// TIA Portal V17 export
// export: Created 2025-03-07T09:19:05.7984013Z, ExportSetting WithDefaults, DisplayName Totally Integrated Automation Portal, DisplayVersion V17 Update 8, DisplayName TIA Portal Openness, DisplayVersion V17 Update 8, DisplayName TIA Portal Version Control Interface, DisplayVersion V17, DisplayName SINAMICS Startdrive Advanced, DisplayVersion V17 SP2, DisplayName SINAMICS Startdrive G110M, G120, G120C, G120D, G120P, G115D, DisplayVersion V17 SP2, DisplayName SINAMICS Startdrive G130, G150, S120, S150, SINAMICS MV, S210, DisplayVersion V17 SP2, DisplayName STEP 7 Professional, DisplayVersion V17 Update 8, DisplayName SINUMERIK ONE STEP 7 Toolbox, DisplayVersion V17 Update 12, DisplayName SINUMERIK 840D sl STEP 7 Toolbox, DisplayVersion V17 Update 12, DisplayName STEP 7 Safety, DisplayVersion V17 Update 6, DisplayName WinCC Advanced, DisplayVersion V17 Update 8
DATA_BLOCK "DB16701_OPC_UA_MASTER_MACHINE"   // DB16701
{ S7_Optimized_Access := 'FALSE' }
VERSION : 0.1
// stored: AutoNumber false, DBAccessibleFromOPCUA true, DBAccessibleFromWebserver true, IsOnlyStoredInLoadMemory false, IsWriteProtectedInAS false
   VAR
      GENERAL { ExternalWritable := 'False'} : Struct
         ID { ExternalWritable := 'False'} : Struct
            LINE { ExternalWritable := 'False'} : Int;   // GENERAL INFORMATION: PRODUCTION LINE IDENTIFICATION
            MACHINE { ExternalWritable := 'False'} : Int;   // GENERAL INFORMATION: PRODUCTION MACHINE IDENTIFICATION
            PLC { ExternalWritable := 'False'} : Int;   // GENERAL INFORMATION: PRODUCTION PLC IDENTIFICATION (POWDER PLC = 1 / MACHINE PLC = 2 / CELL PLC = 3)
         END_STRUCT;
         WORKER { ExternalWritable := 'False'} : Struct
            ID { ExternalWritable := 'False'} : Int;
         END_STRUCT;
         PART_TRACKING { ExternalWritable := 'False'} : Struct
            UNIT_01 { ExternalWritable := 'False'} : Struct
               STA1 { ExternalWritable := 'False'} : Struct
                  DMC { ExternalWritable := 'False'} : Array[0..63] of Char;   // DMC PART NUMBER IN UNIT 01 STATION 1
                  FIXTURE_NUMBER { ExternalWritable := 'False'} : Int;   // FIXTURE NUMBER IN UNIT 01 STATION 1
               END_STRUCT;
               STA2 { ExternalWritable := 'False'} : Struct
                  DMC { ExternalWritable := 'False'} : Array[0..63] of Char;   // DMC PART NUMBER IN UNIT 01 STATION 2
                  FIXTURE_NUMBER { ExternalWritable := 'False'} : Int;   // FIXTURE NUMBER IN UNIT 01 STATION 2
               END_STRUCT;
               STA3 { ExternalWritable := 'False'} : Struct
                  DMC { ExternalWritable := 'False'} : Array[0..63] of Char;   // DMC PART NUMBER IN UNIT 01 STATION 3
                  FIXTURE_NUMBER { ExternalWritable := 'False'} : Int;   // FIXTURE NUMBER IN UNIT 01 STATION 3
               END_STRUCT;
               STA4 { ExternalWritable := 'False'} : Struct
                  DMC { ExternalWritable := 'False'} : Array[0..63] of Char;   // DMC PART NUMBER IN UNIT 01 STATION 4
                  FIXTURE_NUMBER { ExternalWritable := 'False'} : Int;   // FIXTURE NUMBER IN UNIT 01 STATION 4
               END_STRUCT;
            END_STRUCT;
            UNIT_02 { ExternalWritable := 'False'} : Struct
               STA1 { ExternalWritable := 'False'} : Struct
                  DMC { ExternalWritable := 'False'} : Array[0..63] of Char;   // DMC PART NUMBER IN UNIT 02 STATION 1
                  FIXTURE_NUMBER { ExternalWritable := 'False'} : Int;   // FIXTURE NUMBER IN UNIT 02 STATION 1
               END_STRUCT;
               STA2 { ExternalWritable := 'False'} : Struct
                  DMC { ExternalWritable := 'False'} : Array[0..63] of Char;   // DMC PART NUMBER IN UNIT 02 STATION 2
                  FIXTURE_NUMBER { ExternalWritable := 'False'} : Int;   // FIXTURE NUMBER IN UNIT 02 STATION 2
               END_STRUCT;
               STA3 { ExternalWritable := 'False'} : Struct
                  DMC { ExternalWritable := 'False'} : Array[0..63] of Char;   // DMC PART NUMBER IN UNIT 02 STATION 3
                  FIXTURE_NUMBER { ExternalWritable := 'False'} : Int;   // FIXTURE NUMBER IN UNIT 02 STATION 3
               END_STRUCT;
               STA4 { ExternalWritable := 'False'} : Struct
                  DMC { ExternalWritable := 'False'} : Array[0..63] of Char;   // DMC PART NUMBER IN UNIT 02 STATION 4
                  FIXTURE_NUMBER { ExternalWritable := 'False'} : Int;   // FIXTURE NUMBER IN UNIT 02 STATION 4
               END_STRUCT;
            END_STRUCT;
         END_STRUCT;
         SHARED_AIR_EXTRACTION { ExternalWritable := 'False'} : Struct
            INPUT_KELLER_PRESSURE { ExternalWritable := 'False'} : Real;   // MACHINE AIR EXTRACTION INPUT KELLER PRESSURE VALUE (Bar)
            PRESSURE_DIFFERENCE_FILTER { ExternalWritable := 'False'} : Real;   // MACHINE AIR EXTRACTION PRESSURE DIFFERENCE IN FILTER VALUE (Bar)
         END_STRUCT;
      END_STRUCT;
      UNIT_01 { ExternalWritable := 'False'} : Struct
         MACHINE { ExternalWritable := 'False'} : Struct
            PNEUMATIC_STATE { ExternalWritable := 'False'} : Bool;   // UNIT 01 PNEUMATIC STATE: CORRECT WORKING (NO FAULTS)
            TEMPERATURE { ExternalWritable := 'False'} : Struct
               DISC_SURFACE { ExternalWritable := 'False'} : Real;   // UNIT 01 MACHINE TEMPERATURE: DISC SURFACE (ºC)
               AMBIENT_PYROMETER { ExternalWritable := 'False'} : Real;   // UNIT 01 MACHINE TEMPERATURE: AMBIENT PYROMETER (ºC)
               EMISIVITY_CURVE { ExternalWritable := 'False'} : Real;   // UNIT 01 MACHINE TEMPERATURE: EMISIVITY CURVE (¿?¿?¿?¿?¿?)
            END_STRUCT;
            COOLING_SYSTEM { ExternalWritable := 'False'} : Struct
               INPUT_FLOW { ExternalWritable := 'False'} : Real;   // UNIT 01 COOLING SYSTEM INPUT FLOW VALUE (l/min)
               INPUT_TEMPERATURE { ExternalWritable := 'False'} : Real;   // UNIT 01 COOLING SYSTEM INPUT TEMPERATURE VALUE (ºC)
               OUTPUT_FLOW { ExternalWritable := 'False'} : Real;   // UNIT 01 COOLING SYSTEM OUTPUT FLOW VALUE (l/min)
               OUTPUT_TEMPERATURE { ExternalWritable := 'False'} : Real;   // UNIT 01 COOLING SYSTEM OUTPUT TEMPERATURE VALUE (ºC)
               LASER_HEAD_FLOW { ExternalWritable := 'False'} : Real;   // UNIT 01 COOLING SYSTEM LASER HEAD FLOW VALUE (l/min)
               LASER_HEAD_TEMPERATURE { ExternalWritable := 'False'} : Real;   // UNIT 01 COOLING SYSTEM LASER HEAD TEMPERATURE VALUE (ºC)
               LASER_FLOW { ExternalWritable := 'False'} : Real;   // UNIT 01 COOLING SYSTEM LASER FLOW VALUE (l/min)
               LASER_TEMPERATURE { ExternalWritable := 'False'} : Real;   // UNIT 01 COOLING SYSTEM LASER TEMPERATURE VALUE (ºC)
               NOZZLE_FLOW { ExternalWritable := 'False'} : Real;   // UNIT 01 COOLING SYSTEM LASER NOZZLE FLOW VALUE (l/min)
               NOZZLE_TEMPERATURE { ExternalWritable := 'False'} : Real;   // UNIT 01 COOLING SYSTEM LASER NOZZLE TEMPERATURE VALUE (ºC)
               SHIELD_FLOW { ExternalWritable := 'False'} : Real;   // UNIT 01 COOLING SYSTEM SHIELD FLOW VALUE (l/min)
               SHIELD_TEMPERATURE { ExternalWritable := 'False'} : Real;   // UNIT 01 COOLING SYSTEM SHIELD TEMPERATURE VALUE (ºC)
            END_STRUCT;
            AIR_EXTRACTION { ExternalWritable := 'False'} : Struct
               OUTPUT_PRESSURE { ExternalWritable := 'False'} : Real;   // UNIT 01 AIR EXTRACTION OUTPUT PRESSURE VALUE (Bar)
               ST3_PRESSURE { ExternalWritable := 'False'} : Real;   // UNIT 01 STA 3 PRESSURE CONTROL
            END_STRUCT;
            POSITIONS { ExternalWritable := 'False'} : Struct
               CN { ExternalWritable := 'False'} : Struct
                  X13 { ExternalWritable := 'False'} : Real;   // UNIT 01 AXIS X13 POSITION VALUE
                  Z13 { ExternalWritable := 'False'} : Real;   // UNIT 01 AXIS Z13 POSITION VALUE
               END_STRUCT;
               LASER_HEAD { ExternalWritable := 'False'} : Struct
                  RADIAL_ANGLE { ExternalWritable := 'False'} : Bool;   // UNIT 01 LASER HEAD RADIAL ANGLE ADVANCED
                  TANGENTIAL_ANGLE { ExternalWritable := 'False'} : Bool;   // UNIT 01 LASER HEAD TANGENTIAL ANGLE ADVANCED
               END_STRUCT;
            END_STRUCT;
            SPEED { ExternalWritable := 'False'} : Struct
               X13 { ExternalWritable := 'False'} : Real;   // UNIT 01 AXIS X13 SPEED VALUE (mm/min)
               C13 { ExternalWritable := 'False'} : Real;   // UNIT 01 AXIS C13 SPEED VALUE (º/min)
               PROCESS_SETPOINT { ExternalWritable := 'False'} : Real;   // UNIT 01 SPEED PROCESS SETPOINT (mm/min)
            END_STRUCT;
            NOZZLE { ExternalWritable := 'False'} : Struct
               SHIELD_GAS_FLOW { ExternalWritable := 'False'} : Real;   // UNIT 01 SHIELD GAS FLOW VALUE (nl/min)
            END_STRUCT;
         END_STRUCT;
         PROCESS { ExternalWritable := 'False'} : Struct
            STATION_1_RUNNING { ExternalWritable := 'False'} : Bool;   // UNIT 01 CLADDING STATION 1 RUNNING
            STATION_2_RUNNING { ExternalWritable := 'False'} : Bool;   // UNIT 01 CLADDING STATION 2 RUNNING
            STATION_3_RUNNING { ExternalWritable := 'False'} : Bool;   // UNIT 01 CLADDING STATION 3 RUNNING
            STATION_4_RUNNING { ExternalWritable := 'False'} : Bool;   // UNIT 01 CLADDING STATION 4 RUNNING
            LASER_ON { ExternalWritable := 'False'} : Bool;   // UNIT 01 LASER ON
            FIXTURE_SEALING { ExternalWritable := 'False'} : Bool;   // UNIT 01 FIXTURE SEALING CLOSED
         END_STRUCT;
      END_STRUCT;
      UNIT_02 { ExternalWritable := 'False'} : Struct
         MACHINE { ExternalWritable := 'False'} : Struct
            PNEUMATIC_STATE { ExternalWritable := 'False'} : Bool;   // UNIT 02 PNEUMATIC STATE: CORRECT WORKING (NO FAULTS)
            TEMPERATURE { ExternalWritable := 'False'} : Struct
               DISC_SURFACE { ExternalWritable := 'False'} : Real;   // UNIT 02 MACHINE TEMPERATURE: DISC SURFACE (ºC)
               AMBIENT_PYROMETER { ExternalWritable := 'False'} : Real;   // UNIT 02 MACHINE TEMPERATURE: AMBIENT PYROMETER (ºC)
               EMISIVITY_CURVE { ExternalWritable := 'False'} : Real;   // UNIT 02 MACHINE TEMPERATURE: EMISIVITY CURVE (¿?¿?¿?¿?¿?)
            END_STRUCT;
            COOLING_SYSTEM { ExternalWritable := 'False'} : Struct
               INPUT_FLOW { ExternalWritable := 'False'} : Real;   // UNIT 02 COOLING SYSTEM INPUT FLOW VALUE (l/min)
               INPUT_TEMPERATURE { ExternalWritable := 'False'} : Real;   // UNIT 02 COOLING SYSTEM INPUT TEMPERATURE VALUE (ºC)
               OUTPUT_FLOW { ExternalWritable := 'False'} : Real;   // UNIT 02 COOLING SYSTEM OUTPUT FLOW VALUE (l/min)
               OUTPUT_TEMPERATURE { ExternalWritable := 'False'} : Real;   // UNIT 02 COOLING SYSTEM OUTPUT TEMPERATURE VALUE (ºC)
               LASER_HEAD_FLOW { ExternalWritable := 'False'} : Real;   // UNIT 02 COOLING SYSTEM LASER HEAD FLOW VALUE (l/min)
               LASER_HEAD_TEMPERATURE { ExternalWritable := 'False'} : Real;   // UNIT 02 COOLING SYSTEM LASER HEAD TEMPERATURE VALUE (ºC)
               LASER_FLOW { ExternalWritable := 'False'} : Real;   // UNIT 02 COOLING SYSTEM LASER FLOW VALUE (l/min)
               LASER_TEMPERATURE { ExternalWritable := 'False'} : Real;   // UNIT 02 COOLING SYSTEM LASER TEMPERATURE VALUE (ºC)
               NOZZLE_FLOW { ExternalWritable := 'False'} : Real;   // UNIT 02 COOLING SYSTEM LASER NOZZLE FLOW VALUE (l/min)
               NOZZLE_TEMPERATURE { ExternalWritable := 'False'} : Real;   // UNIT 02 COOLING SYSTEM LASER NOZZLE TEMPERATURE VALUE (ºC)
               SHIELD_FLOW { ExternalWritable := 'False'} : Real;   // UNIT 02 COOLING SYSTEM SHIELD FLOW VALUE (l/min)
               SHIELD_TEMPERATURE { ExternalWritable := 'False'} : Real;   // UNIT 02 COOLING SYSTEM SHIELD TEMPERATURE VALUE (ºC)
            END_STRUCT;
            AIR_EXTRACTION { ExternalWritable := 'False'} : Struct
               OUTPUT_PRESSURE { ExternalWritable := 'False'} : Real;   // UNIT 02 AIR EXTRACTION OUTPUT PRESSURE VALUE (Bar)
               ST3_PRESSURE { ExternalWritable := 'False'} : Real;   // UNIT 02 STA 3 PRESSURE CONTROL
            END_STRUCT;
            POSITIONS { ExternalWritable := 'False'} : Struct
               CN { ExternalWritable := 'False'} : Struct
                  X23 { ExternalWritable := 'False'} : Real;   // UNIT 02 AXIS X23 POSITION VALUE
                  Z23 { ExternalWritable := 'False'} : Real;   // UNIT 02 AXIS Z23 POSITION VALUE
               END_STRUCT;
               LASER_HEAD { ExternalWritable := 'False'} : Struct
                  RADIAL_ANGLE { ExternalWritable := 'False'} : Bool;   // UNIT 02 LASER HEAD RADIAL ANGLE ADVANCED
                  TANGENTIAL_ANGLE { ExternalWritable := 'False'} : Bool;   // UNIT 02 LASER HEAD TANGENTIAL ANGLE ADVANCED
               END_STRUCT;
            END_STRUCT;
            SPEED { ExternalWritable := 'False'} : Struct
               X23 { ExternalWritable := 'False'} : Real;   // UNIT 02 AXIS X23 SPEED VALUE (mm/min)
               C23 { ExternalWritable := 'False'} : Real;   // UNIT 02 AXIS C23 SPEED VALUE (º/min)
               PROCESS_SETPOINT { ExternalWritable := 'False'} : Real;   // UNIT 02 SPEED PROCESS SETPOINT (mm/min)
            END_STRUCT;
            NOZZLE { ExternalWritable := 'False'} : Struct
               SHIELD_GAS_FLOW { ExternalWritable := 'False'} : Real := 0.0;   // UNIT 02 SHIELD GAS FLOW VALUE (nl/min)
            END_STRUCT;
         END_STRUCT;
         PROCESS { ExternalWritable := 'False'} : Struct
            STATION_1_RUNNING { ExternalWritable := 'False'} : Bool;   // UNIT 02 CLADDING STATION 1 RUNNING
            STATION_2_RUNNING { ExternalWritable := 'False'} : Bool;   // UNIT 02 CLADDING STATION 2 RUNNING
            STATION_3_RUNNING { ExternalWritable := 'False'} : Bool;   // UNIT 02 CLADDING STATION 3 RUNNING
            STATION_4_RUNNING { ExternalWritable := 'False'} : Bool;   // UNIT 02 CLADDING STATION 4 RUNNING
            LASER_ON { ExternalWritable := 'False'} : Bool;   // UNIT 02 LASER ON
            FIXTURE_SEALING { ExternalWritable := 'False'} : Bool;   // UNIT 02 FIXTURE SEALING CLOSED
         END_STRUCT;
      END_STRUCT;
   END_VAR
BEGIN
END_DATA_BLOCK
